FUNCTION_BLOCK fbPulser
VAR_INPUT
	bInRun:		BOOL;	(*Enables the pulsing output*)
	tInTimeOn:	TIME;	(*Amount of time output is turned on each period*)
	tInTimeOff:	TIME;	(*Amount of time output is off each period*)
	iInNumPulses: INT;	(*Number of pulses to output (0 for infinite)*)
END_VAR
VAR_OUTPUT
	bOutPulse:	BOOL;	(*The pulsing output*)
	bOutDone:	BOOL;	(*Pulsing complete, iNumPulses achieved*)
	iOutCount:	INT;	(*Current number of pulses complete*)

END_VAR
VAR
	rTrigbRun:R_TRIG;
	nState: INT;
	tonTimerOn:TON;
	tonTimerOff:TON;
END_VAR

rTrigbRun(CLK:=bInRun , Q=> );

//When a new run command is issued the pulsing sequence is restarted
IF rTrigbRun.Q THEN
	nState:=10;
END_IF

CASE nstate OF
	0:
		bOutPulse:=0;
		iOutCount:=0;
		
	10:
		bOutPulse:=1;
		IF NOT(bInRun) OR bOutDone THEN
			nState:=0;
		ELSIF tonTimerOn.Q THEN
			iOutCount:=iOutCount+1;
			nState:=20;
		END_IF	
	20:
		bOutPulse:=0;
		IF NOT(bInRun) OR bOutDone THEN
			nState:=0;
		ELSIF tonTimerOff.Q THEN
			nState:=10;
		END_IF	
		
END_CASE

bOutDone:=(iOutCount>=iInNumPulses) AND NOT(iInNumPulses=0);  // run infinitely if inumpulse=0
tonTimerOn(IN:=(nState=10) , PT:=tInTimeOn , Q=> , ET=> );	  // time in state 10 -- time pulse on	
tonTimerOff(IN:=(nState=20) , PT:=tInTimeOff , Q=> , ET=> );	  // time in state 20 -- time pulse off

END_FUNCTION_BLOCK

(* stored: Version 1.1.0.1, ProductVersion 3.1.4024.11
   POU fbPulser: Id {4768702a-1f4e-47c6-a6fa-2989d4e8390c}, SpecialFunc None *)
